(* IEC 61131-3 sources: lasal-git-demo/CPU/LasalDemoProject/Class/DI200, 1 file *)

(* ---- DI200.st ---- *)
#define DEVICE_ID_DI200 1001

(*!
<Class
	Name               = "DI200"
	Revision           = "1.42"
	RealtimeTask       = "false"
	CyclicTask         = "false"
	BackgroundTask     = "false"
	Sigmatek           = "true"
	OSInterface        = "false"
	HighPriority       = "false"
	Automatic          = "false"
	UpdateMode         = "Prescan"
	IconPath           = ".\Class\s-dias.ico"
	SharedCommandTable = "true"
	Objectsize         = "(398,120)"
	Comment            = "This hardware class is used to control the DI200 hardware module with 20 digital inputs.">
	<Channels>
		<Server Name="Input1" Visualized="true" Initialize="false" WriteProtected="true" Retentive="false" Comment="Input 1 value"/>
		<Server Name="Input10" Visualized="true" Initialize="false" WriteProtected="true" Retentive="false" Comment="Input 10 value"/>
		<Server Name="Input11" Visualized="true" Initialize="false" WriteProtected="true" Retentive="false" Comment="Input 11 value"/>
		<Server Name="Input12" Visualized="true" Initialize="false" WriteProtected="true" Retentive="false" Comment="Input 12 value"/>
		<Server Name="Input13" Visualized="true" Initialize="false" WriteProtected="true" Retentive="false" Comment="Input 13 value"/>
		<Server Name="Input14" Visualized="true" Initialize="false" WriteProtected="true" Retentive="false" Comment="Input 14 value"/>
		<Server Name="Input15" Visualized="true" Initialize="false" WriteProtected="true" Retentive="false" Comment="Input 15 value"/>
		<Server Name="Input16" Visualized="true" Initialize="false" WriteProtected="true" Retentive="false" Comment="Input 16 value"/>
		<Server Name="Input17" Visualized="true" Initialize="false" WriteProtected="true" Retentive="false" Comment="Input 17 value"/>
		<Server Name="Input18" Visualized="true" Initialize="false" WriteProtected="true" Retentive="false" Comment="Input 18 value"/>
		<Server Name="Input19" Visualized="true" Initialize="false" WriteProtected="true" Retentive="false" Comment="Input 19 value"/>
		<Server Name="Input2" Visualized="true" Initialize="false" WriteProtected="true" Retentive="false" Comment="Input 2 value"/>
		<Server Name="Input20" Visualized="true" Initialize="false" WriteProtected="true" Retentive="false" Comment="Input 20 value"/>
		<Server Name="Input3" Visualized="true" Initialize="false" WriteProtected="true" Retentive="false" Comment="Input 3 value"/>
		<Server Name="Input4" Visualized="true" Initialize="false" WriteProtected="true" Retentive="false" Comment="Input 4 value"/>
		<Server Name="Input5" Visualized="true" Initialize="false" WriteProtected="true" Retentive="false" Comment="Input 5 value"/>
		<Server Name="Input6" Visualized="true" Initialize="false" WriteProtected="true" Retentive="false" Comment="Input 6 value"/>
		<Server Name="Input7" Visualized="true" Initialize="false" WriteProtected="true" Retentive="false" Comment="Input 7 value"/>
		<Server Name="Input8" Visualized="true" Initialize="false" WriteProtected="true" Retentive="false" Comment="Input 8 value"/>
		<Server Name="Input9" Visualized="true" Initialize="false" WriteProtected="true" Retentive="false" Comment="Input 9 value"/>
		<Server Name="InputDouble" Visualized="true" Initialize="false" WriteProtected="true" Retentive="false" Comment="Bit 0 to 19 ... Input 1 to 20"/>
	</Channels>
	<RevDoku>
		<Owner Company="Sigmatek" Author="BeiWol"/>
		<Dokumentation Revision="1.42" Date="12.08.2019" Author="LazJos" Company="Sigmatek" Description="Added support for HWAlarms."/>
		<Dokumentation Revision="1.41" Date="09.01.2019" Author="FurDom" Company="Sigmatek" Description="Added function for Spi Write in SdiasBase class."/>
		<Dokumentation Revision="1.40" Date="08.06.2018" Author="RamAnd" Company="Sigmatek" Description="LASAL Hardware Description (.lhd) file has been updated."/>
		<Dokumentation Revision="1.39" Date="16.05.2017" Author="RamAnd" Company="Sigmatek" Description="When adding an SDO (i.e. via ReadSPIData) from background priority it was possible that the adding process got interrupted by receiving the answer to this SDO which is handled in cyclic priority. In the error case the answer was unexpected and therefore ignored. Then the class signals a timeout while waiting for the answer, which already arrived before waiting for it. Added mutex and changed instruction order to prevent this error."/>
		<Dokumentation Revision="1.38" Date="12.07.2016" Author="SeiChr" Company="Sigmatek" Description="Added Values for the total Current calculation. SA 31571"/>
		<Dokumentation Revision="1.37" Date="01.03.2016" Author="EisMic" Company="Sigmatek" Description="Corrected BoundExceed Error in base class at Write method of LEDControl Server when Place = LSL_DEACTIVATED."/>
		<Dokumentation Revision="1.36" Date="17.06.2015" Author="EisMic" Company="Sigmatek" Description="The servers FPGAVersion, SerialNo, Device ID and status and input servers are now not reset anymore when the module is disconnected."/>
		<Dokumentation Revision="1.35" Date="16.04.2015" Author="EisMic&#13;&#10;LanSte" Company="Sigmatek" Description="Added support for visualisation in graphical hardware editor.&#13;&#10;Added support for calculating resources for graphical hardware editor."/>
		<Dokumentation Revision="1.34" Date="17.03.2015" Author="RamAnd" Company="Sigmatek" Description="Added HW Version for sdias clients."/>
		<Dokumentation Revision="1.33" Date="11.02.2015" Author="PieSte" Company="Sigmatek" Description="Corrected read spi data for hardwaretree in methode GetSPIDataFromID from baseclass."/>
		<Dokumentation Revision="1.32" Date="18.11.2014" Author="PieSte" Company="Sigmatek" Description="Added possibility  to read more data from spi flash then one sdo access.&#13;&#10;Set methode GetDeviceID to global.&#13;&#10;Add methode to calculate checksum of spi flash."/>
		<Dokumentation Revision="1.31" Date="04.07.2014" Author="EisMic" Company="Sigmatek" Description="Added support for reading hardware diagnosis and hardwaretree entry."/>
		<Dokumentation Revision="1.30" Date="20.01.2014" Author="PieSte" Company="Sigmatek" Description="Read Client Required and Place in Init SdiasBase"/>
		<Dokumentation Revision="1.20" Date="05.12.2013" Author="RamAnd" Company="Sigmatek" Description="Changed login mechanism to sdias manager class to be independent of bus accesses."/>
		<Dokumentation Revision="1.10" Date="01.08.2013" Author="ObeChr" Company="Sigmatek" Description="Modified Clients / Server / Comments&#13;&#10;The class now also shows the FPGA Version on a new Server.&#13;&#10;In the first realtime cycles the classes showed _ClassOk, but there was no actual IO information. Now the ClassState of SDIAS Clients is stored temporary during init and shown at the server after init."/>
		<Dokumentation Revision="1.0" Date="18.07.2013" Author="RamAnd" Company="Sigmatek" Description="First library version"/>
	</RevDoku>
	<Network Name="DI200">
		<!-- List of Components in this network -->
		<Components>
			<Object
				Name       = "_base"
				Class      = "SdiasBase"
				Position   = "(218,120)"
				Visualized = "true">
				<Channels>
					<Server Name="ClassState"/>
					<Server Name="DeviceID"/>
					<Server Name="FPGAVersion"/>
					<Server Name="HwVersion"/>
					<Server Name="LEDControl" Value="0"/>
					<Server Name="RetryCounter"/>
					<Server Name="SDOState"/>
					<Server Name="SerialNo"/>
					<Client Name="Place" Value="0"/>
					<Client Name="Required" Value="1"/>
					<Client Name="SdiasIn"/>
					<Client Name="ToStdLib"/>
				</Channels>
			</Object>
		</Components>
		<Comments>
		</Comments>
		<!-- List of Connections in this network -->
		<Connections>
			<Connection Source="this.ClassState" Destination="_base.ClassState" Vertices="(804,210),(632,210),"/>
			<Connection Source="this.DeviceID" Destination="_base.DeviceID" Vertices="(804,270),(632,270),"/>
			<Connection Source="this.SerialNo" Destination="_base.SerialNo" Vertices="(804,450),(632,450),"/>
			<Connection Source="this.RetryCounter" Destination="_base.RetryCounter" Vertices="(804,510),(632,510),"/>
			<Connection Source="_base.SdiasIn" Destination="this.SdiasIn" Vertices="(218,210),(38,210),"/>
			<Connection Source="_base.Place" Destination="this.Place" Vertices="(218,270),(38,270),"/>
			<Connection Source="_base.Required" Destination="this.Required" Vertices="(218,330),(38,330),"/>
			<Connection Source="this.LEDControl" Destination="_base.LEDControl" Vertices="(804,570),(632,570),"/>
			<Connection Source="this.FPGAVersion" Destination="_base.FPGAVersion" Vertices="(804,330),(632,330),"/>
			<Connection Source="this.HwVersion" Destination="_base.HwVersion" Vertices="(804,390),(632,390),"/>
		</Connections>
		<!-- Headerfiles -->
		<Options>
		</Options>
	</Network>
</Class>
*)
#pragma using SdiasBase

DI200 : CLASS
: SdiasBase
  //Servers:
	Input1 	: SvrCh_DINT;
	Input2 	: SvrCh_DINT;
	Input3 	: SvrCh_DINT;
	Input4 	: SvrCh_DINT;
	Input5 	: SvrCh_DINT;
	Input6 	: SvrCh_DINT;
	Input7 	: SvrCh_DINT;
	Input8 	: SvrCh_DINT;
	Input9 	: SvrCh_DINT;
	Input10 	: SvrCh_DINT;
	Input11 	: SvrCh_DINT;
	Input12 	: SvrCh_DINT;
	Input13 	: SvrCh_DINT;
	Input14 	: SvrCh_DINT;
	Input15 	: SvrCh_DINT;
	Input16 	: SvrCh_DINT;
	Input17 	: SvrCh_DINT;
	Input18 	: SvrCh_DINT;
	Input19 	: SvrCh_DINT;
	Input20 	: SvrCh_DINT;
	InputDouble 	: SvrCh_BDINT;
  //Clients:
  //Variables:
		pReadData 	: ^DINT;
  //Functions:
				//! <Function Comment="Realtime Update Methode which runs in PreScan." Name="UpdateRt"/>
	FUNCTION VIRTUAL GLOBAL UpdateRt;
				//! <Function Comment="Methode is called if this Module gets connected." Name="ConnectEvent"/>
	FUNCTION VIRTUAL GLOBAL ConnectEvent;
				//! <Function Comment="Methode is called if this Module gets disconnected." Name="DisconnectEvent"/>
	FUNCTION VIRTUAL GLOBAL DisconnectEvent;
				//! <Function Comment="This Methode should is used, to check the DeviceID of the Module." Name="CheckDeviceID"/>
	FUNCTION VIRTUAL GLOBAL CheckDeviceID
		VAR_INPUT
			udID2Check 	: UDINT;			//! <Variable Comment="Device ID of connected Module." Name="CheckDeviceID.udID2Check"/>
		END_VAR
		VAR_OUTPUT
			bIsOK 	: BOOL;			//! <Variable Comment="FALSE = Wrong DeviceID for Module&#13;&#10;TRUE  = DeviceID of Module is correct" Name="CheckDeviceID.bIsOK"/>
		END_VAR;

	FUNCTION VIRTUAL GetTaskCfg
		VAR_OUTPUT
			TaskCfg 	: BDINT;			//! <Variable Comment="Select which tasks will be available for this module:&#13;&#10;Bit0..Realtime PreScan&#13;&#10;Bit1..Realtime PostScan&#13;&#10;Bit2..Cyclic&#13;&#10;&#13;&#10;e.g. if only realtime postscan is needed:&#13;&#10;2#010" Name="GetTaskCfg.TaskCfg"/>
		END_VAR;

	FUNCTION VIRTUAL GetDeviceID
		VAR_OUTPUT
			output 	: UDINT;
		END_VAR;
  //Tables:
	FUNCTION @STD
		VAR_OUTPUT
			ret_code	: CONFSTATES;
		END_VAR;
	FUNCTION GLOBAL TAB @CT_;
END_CLASS;

FUNCTION VIRTUAL GLOBAL DI200::UpdateRt
  VAR
    inputMask : DINT;
    newInputs : DINT;
    pInputSrv : ^DINT;
  END_VAR

  newInputs := pReadData^;
  InputMask := InputDouble$DINT xor newInputs; //old Input xor new Input (to see changes)

  if InputMask <> 0 then

    InputDouble$DINT  := newInputs;
    pInputSrv         :=#Input1.Ddata;

    repeat
      if InputMask and 1 then
        pInputSrv^ := newInputs and 1;
      end_if;
      inputMask := inputMask shr 1;
      newInputs := newInputs shr 1;
      pInputSrv += sizeof(SvrCh);
    until inputMask = 0 end_repeat;

  end_if;

END_FUNCTION

FUNCTION VIRTUAL GLOBAL DI200::CheckDeviceID
	VAR_INPUT
		udID2Check 	: UDINT;
	END_VAR
	VAR_OUTPUT
		bIsOK 	: BOOL;
	END_VAR

  //look if it is right hardware
	if ( udID2Check <> DEVICE_ID_DI200 ) then
		bIsOK := FALSE;
	else
    bIsOK := TRUE;
	end_if;

END_FUNCTION

FUNCTION VIRTUAL GLOBAL DI200::ConnectEvent

  // start the accesses on the SDIAS (initialize the control byte in the DPRAM)
  if DefaultAccesses.ReadAccess.pControlByte then
    pReadData := DefaultAccesses.ReadAccess.pData$^DINT;

    DefaultAccesses.ReadAccess.pControlByte^.EnableDO := TRUE;
  else
    eInitState := _DOHandleInvalid;
    return;
  end_if;

  // module is ok
  eInitState := _ClassOk;

END_FUNCTION

FUNCTION VIRTUAL GLOBAL DI200::DisconnectEvent

  // reset general module information shown on servers
  SdiasBase::DisconnectEvent();

END_FUNCTION

FUNCTION VIRTUAL DI200::GetTaskCfg
	VAR_OUTPUT
		TaskCfg 	: BDINT;
	END_VAR

  TaskCfg := SDIAS_TASK_MASK_RT_PRE;

END_FUNCTION

FUNCTION VIRTUAL DI200::GetDeviceID
	VAR_OUTPUT
		output 	: UDINT;
	END_VAR

  output := DEVICE_ID_DI200;

END_FUNCTION
